TYPE TcaWorkpiecePlaceConfig EXTENDS ST_ComboboxEntry:
STRUCT
	
END_STRUCT
END_TYPE

(* stored: Version 1.1.0.1
   DUT TcaWorkpiecePlaceConfig: Id {85a84314-a765-46c5-83f4-70b267464807} *)
